// TIA Portal project "练习_V17" (V17)

(* hardware
DEVICE "S7-1200 station_1"  S7-1200 Station
   slot 0: "Rack_0"  S7-1200 Rack  Rack  V1.0
   slot 1: "PLC_1"  CPU 1215C DC/DC/DC  6ES7 215-1AG40-0XB0  V4.2
*)

// ===== PLC "PLC_1"  CPU 1215C DC/DC/DC =====

VAR_GLOBAL   // PLC tag table "默认变量表"
   "Q0.2" AT %Q0.2 : Bool;
   "Q0.3" AT %Q0.3 : Bool;
   "Q0.4" AT %Q0.4 : Bool;
   "Q0.5" AT %Q0.5 : Bool;
   "M2.4" AT %M2.4 : Bool;
   "M2.5" AT %M2.5 : Bool;
   "M2.6" AT %M2.6 : Bool;
   "M2.7" AT %M2.7 : Bool;
   "M3.0" AT %M3.0 : Bool;
   "M3.1" AT %M3.1 : Bool;
   "M3.2" AT %M3.2 : Bool;
   "M3.3" AT %M3.3 : Bool;
   "M2.0" AT %M2.0 : Bool;
   "M2.1" AT %M2.1 : Bool;
   "M2.2" AT %M2.2 : Bool;
   "M2.3" AT %M2.3 : Bool;
   "Q0.0" AT %Q0.0 : Bool;
   "Q0.1" AT %Q0.1 : Bool;
   "MD100" AT %MD100 : Time;
   "MD104" AT %MD104 : Time;
   "MD10" AT %MD10 : Real;
   "MD14" AT %MD14 : Real;
   "MD18" AT %MD18 : Real;
   "MD22" AT %MD22 : Real;
   "MD26" AT %MD26 : Real;
   "System_Byte" AT %MB1 : Byte;
   "FirstScan" AT %M1.0 : Bool;
   "DiagStatusUpdate" AT %M1.1 : Bool;
   "AlwaysTRUE" AT %M1.2 : Bool;
   "AlwaysFALSE" AT %M1.3 : Bool;
   "Clock_Byte" AT %MB0 : Byte;
   "Clock_10Hz" AT %M0.0 : Bool;
   "Clock_5Hz" AT %M0.1 : Bool;
   "Clock_2.5Hz" AT %M0.2 : Bool;
   "Clock_2Hz" AT %M0.3 : Bool;
   "Clock_1.25Hz" AT %M0.4 : Bool;
   "Clock_1Hz" AT %M0.5 : Bool;
   "Clock_0.625Hz" AT %M0.6 : Bool;
   "Clock_0.5Hz" AT %M0.7 : Bool;
   "MW30" AT %MW30 : UInt;
   "MW32" AT %MW32 : UInt;
   "MW34" AT %MW34 : UInt;
   "MW36" AT %MW36 : Int;
   "MW38" AT %MW38 : Int;
   "MW40" AT %MW40 : Int;
   "轴_3_方向" AT %Q0.6 : Bool;
   "轴_4_方向" AT %Q0.7 : Bool;
END_VAR

TYPE "运动轴"
   STRUCT
      输入 : Struct
         "IN:轴使能" : Bool := false;
         "IN:轴复位" : Bool := false;
         "IN:轴回原" : Bool := false;
         "IN:停轴" : Bool := false;
         "IN:绝对定位开" : Bool := false;
         "IN:相对定位开" : Bool := false;
         "IN:手动向前" : Bool := false;
         "IN:手动向后" : Bool := false;
         "IN:绝对目标位置" : Real := 0.0;
         "IN:相对目标位置" : Real := 0.0;
         "IN:绝对定位速度" : Real := 0.0;
         "IN:相对定位速度" : Real := 0.0;
         "IN:手动速度" : Real := 0.0;
      END_STRUCT;
      输出 : Struct
         轴使能状态 : Bool := false;
         轴错误 : Bool := false;
         轴复位完成 : Bool := false;
         轴回原完成 : Bool := false;
         轴回原中 : Bool := false;
         轴回原完成通知 : Bool := false;
         轴暂停中 : Bool := false;
         轴绝对定位完成 : Bool := false;
         轴绝对定位中 : Bool := false;
         轴相对定位完成 : Bool := false;
         轴相对定位中 : Bool := false;
         轴手动行走完成 : Bool := false;
         轴手动行走中 : Bool := false;
         轴错误代码 : Word := 16#0;
         轴错误详情 : Word := 16#0;
      END_STRUCT;
   END_STRUCT;
END_TYPE

// folder: 10-运动控制

DATA_BLOCK "轴控制_DB"   // DB13
{ S7_Optimized_Access := 'TRUE' }
VERSION : 0.1
// stored: InstanceOfName 轴控制
"轴控制"
BEGIN
END_DATA_BLOCK

DATA_BLOCK "运动轴数据"   // DB14
{ S7_Optimized_Access := 'FALSE' }
VERSION : 0.1
   VAR
      轴1 : "运动轴";
      轴2 : "运动轴";
      轴3 : "运动轴";
      轴4 : "运动轴";
   END_VAR
BEGIN
END_DATA_BLOCK

// folder: 20-报警

DATA_BLOCK "报警模块_DB"   // DB22
{ S7_Optimized_Access := 'TRUE' }
VERSION : 0.1
// stored: InstanceOfName 报警灯
"报警灯"
BEGIN
END_DATA_BLOCK

// folder: (top level)

DATA_BLOCK "轴_1"   // DB1, Motion_DB
{ S7_Optimized_Access := 'TRUE' }
AUTHOR : SIMATIC
FAMILY : BasicMC
NAME : TO_PosAx
VERSION : 6.0
// stored: InstanceOfName TO_PositioningAxis
"TO_PositioningAxis"
BEGIN
   // Axis.OnlinePtoModeCU = 16#0000_0002
   // Axis.DirectionOutputEnabledCU = TRUE
   // Axis.SelectedChannel2EnumCU = %Q0.4
   // Axis.SelectedChannel1EnumCU = %Q0.0
   // Pulse.MinDeltaDeltaFrequencyCU = 0.004
   // Pulse.MaxDeltaDeltaFrequencyCU = 1.0E+10
   // Pulse.MinDeltaFrequencyCU = 0.005
   // Pulse.MaxDeltaFrequencyCU = 9.5E+9
   // Pulse.MinFrequencyCU = 1.0
   // Pulse.MaxFrequencyCU = 100000.0
   // Pulse.OutputSourceCU = 16#0000_0000
   // Axis.SelectPTO = 0
END_DATA_BLOCK

DATA_BLOCK "轴_2"   // DB2, Motion_DB
{ S7_Optimized_Access := 'TRUE' }
AUTHOR : SIMATIC
FAMILY : BasicMC
NAME : TO_PosAx
VERSION : 6.0
// stored: InstanceOfName TO_PositioningAxis
"TO_PositioningAxis"
BEGIN
   // Axis.OnlinePtoModeCU = 16#0000_0002
   // Axis.DirectionOutputEnabledCU = TRUE
   // Axis.SelectedChannel2EnumCU = %Q0.5
   // Axis.SelectedChannel1EnumCU = %Q0.1
   // Pulse.MinDeltaDeltaFrequencyCU = 0.004
   // Pulse.MaxDeltaDeltaFrequencyCU = 1.0E+10
   // Pulse.MinDeltaFrequencyCU = 0.005
   // Pulse.MaxDeltaFrequencyCU = 9.5E+9
   // Pulse.MinFrequencyCU = 1.0
   // Pulse.MaxFrequencyCU = 100000.0
   // Pulse.OutputSourceCU = 16#0000_0000
   // Axis.SelectPTO = 1
   // Axis.OnlinePtoIndexCU = 1
END_DATA_BLOCK

DATA_BLOCK "轴_3"   // DB3, Motion_DB
{ S7_Optimized_Access := 'TRUE' }
AUTHOR : SIMATIC
FAMILY : BasicMC
NAME : TO_PosAx
VERSION : 6.0
// stored: InstanceOfName TO_PositioningAxis
"TO_PositioningAxis"
BEGIN
   // Axis.OnlinePtoModeCU = 16#0000_0002
   // Axis.DirectionOutputEnabledCU = TRUE
   // Axis.SelectedChannel2EnumCU = %Q0.6
   // Axis.SelectedChannel1EnumCU = %Q0.2
   // Pulse.MinDeltaDeltaFrequencyCU = 0.004
   // Pulse.MaxDeltaDeltaFrequencyCU = 1.0E+10
   // Pulse.MinDeltaFrequencyCU = 0.005
   // Pulse.MaxDeltaFrequencyCU = 9.5E+9
   // Pulse.MinFrequencyCU = 1.0
   // Pulse.MaxFrequencyCU = 100000.0
   // Pulse.OutputSourceCU = 16#0000_0000
   // Axis.SelectPTO = 2
   // Axis.OnlinePtoIndexCU = 2
END_DATA_BLOCK

DATA_BLOCK "轴_4"   // DB4, Motion_DB
{ S7_Optimized_Access := 'TRUE' }
AUTHOR : SIMATIC
FAMILY : BasicMC
NAME : TO_PosAx
VERSION : 6.0
// stored: InstanceOfName TO_PositioningAxis
"TO_PositioningAxis"
BEGIN
   // Axis.OnlinePtoModeCU = 16#0000_0002
   // Axis.DirectionOutputEnabledCU = TRUE
   // Axis.SelectedChannel2EnumCU = %Q0.7
   // Axis.SelectedChannel1EnumCU = %Q0.3
   // Pulse.MinDeltaDeltaFrequencyCU = 0.004
   // Pulse.MaxDeltaDeltaFrequencyCU = 1.0E+10
   // Pulse.MinDeltaFrequencyCU = 0.005
   // Pulse.MaxDeltaFrequencyCU = 9.5E+9
   // Pulse.MinFrequencyCU = 1.0
   // Pulse.MaxFrequencyCU = 100000.0
   // Pulse.OutputSourceCU = 16#0000_0000
   // Axis.SelectPTO = 3
   // Axis.OnlinePtoIndexCU = 3
END_DATA_BLOCK

ORGANIZATION_BLOCK "Main"   // OB1, LAD, ProgramCycle
TITLE = "Main Program Sweep (Cycle)"
{ S7_Optimized_Access := 'TRUE' }
VERSION : 0.1
   VAR_INPUT
      Initial_Call : Bool;   // Initial call of this OB
      Remanence : Bool;   // =True, if remanent data are available
   END_VAR
BEGIN

REGION Network 2
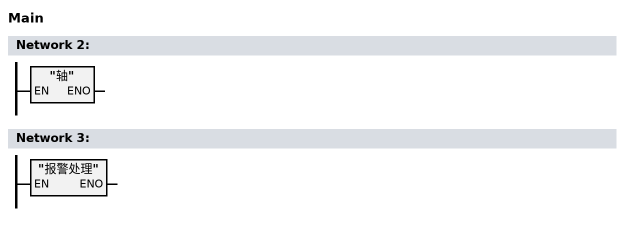
   RUNG wire#powerrail
      "轴"()
   END_RUNG
   // the same network as SCL:
   "轴"();
END_REGION

REGION Network 3
   RUNG wire#powerrail
      "报警处理"()
   END_RUNG
   // the same network as SCL:
   "报警处理"();
END_REGION
END_ORGANIZATION_BLOCK

// folder: 10-运动控制

FUNCTION_BLOCK "轴底层"   // FB11, LAD
{ S7_Optimized_Access := 'TRUE' }
VERSION : 0.1
   VAR_INPUT
      "IN:轴使能" : Bool;
      "IN:轴复位" : Bool;
      "IN:轴回原" : Bool;
      "IN:停轴" : Bool;
      "IN:绝对定位开" : Bool;
      "IN:相对定位开" : Bool;
      "IN:手动向前" : Bool;
      "IN:手动向后" : Bool;
      "IN:绝对目标位置" : Real;
      "IN:相对目标位置" : Real;
      "IN:绝对定位速度" : Real;
      "IN:相对定位速度" : Real;
      "IN:手动速度" : Real;
   END_VAR
   VAR_OUTPUT
      轴使能状态 : Bool;
      轴错误 : Bool;
      轴复位完成 : Bool;
      轴回原完成 : Bool;
      轴回原中 : Bool;
      轴回原完成通知 : Bool;
      轴暂停中 : Bool;
      轴绝对定位完成 : Bool;
      轴绝对定位中 : Bool;
      轴相对定位完成 : Bool;
      轴相对定位中 : Bool;
      轴手动行走完成 : Bool;
      轴手动行走中 : Bool;
      轴错误代码 : Word;
      轴错误详情 : Word;
   END_VAR
   VAR_IN_OUT
      轴 : TO_Axis;
      速度轴 : TO_SpeedAxis;
      定位轴 : TO_PositioningAxis;
   END_VAR
   VAR
      轴使能块 : MC_Power;
      轴复位块 : MC_Reset;
      轴回原块 : MC_Home;
      轴停止块 : MC_Halt;
      轴绝对定位块 : MC_MoveAbsolute;
      轴相对定位快 : MC_MoveRelative;
      轴手动 : MC_MoveJog;
      错误1 : Bool;
      错误2 : Bool;
      错误3 : Bool;
      错误4 : Bool;
      错误5 : Bool;
      错误6 : Bool;
      错误7 : Bool;
   END_VAR
BEGIN

REGION Network 1: 使能
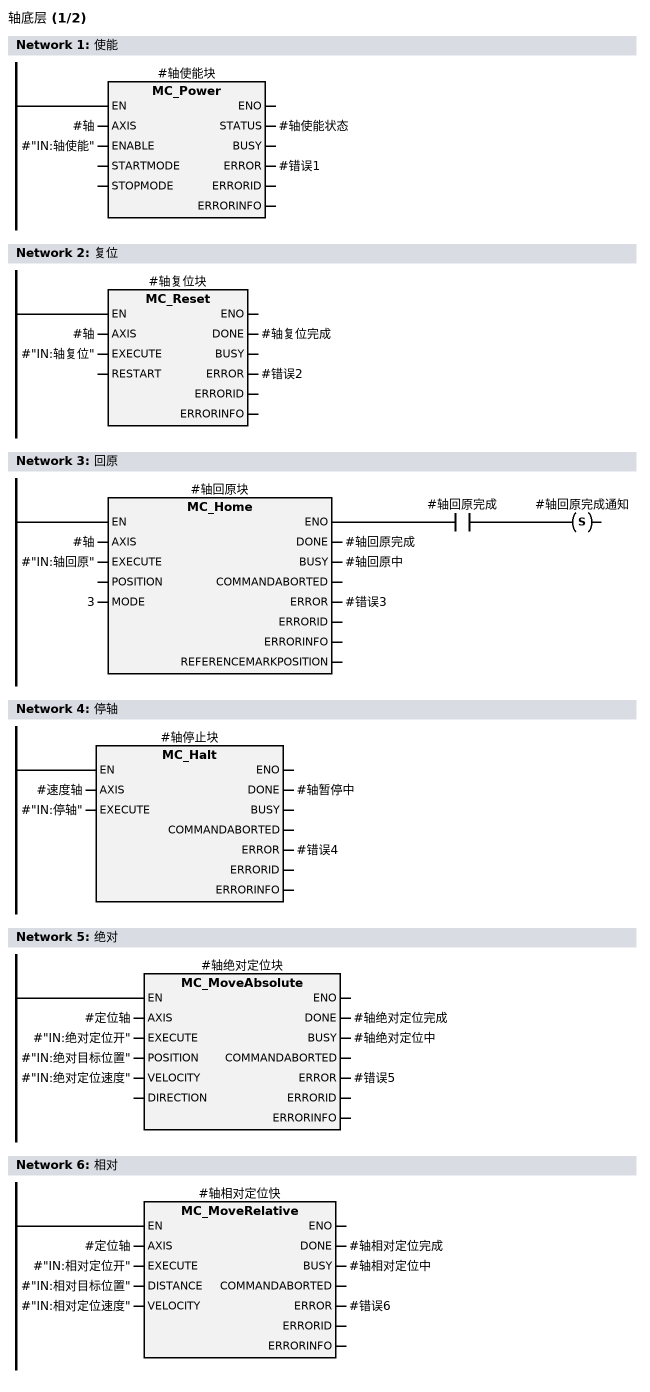
   #轴使能块(Axis := #轴, Enable := #"IN:轴使能", Status => #轴使能状态, Error => #错误1);   // MC_Power
END_REGION

REGION Network 2: 复位
   #轴复位块(Axis := #轴, Execute := #"IN:轴复位", Done => #轴复位完成, Error => #错误2);   // MC_Reset
END_REGION

REGION Network 3: 回原
   // ENO of a box is taken as its EN; it also drops when the box reports an error
   #轴回原块(Axis := #轴, Execute := #"IN:轴回原", Mode := 3, Done => #轴回原完成, Busy => #轴回原中, Error => #错误3);   // MC_Home
   IF #轴回原完成 THEN #轴回原完成通知 := TRUE; END_IF;
END_REGION

REGION Network 4: 停轴
   #轴停止块(Axis := #速度轴, Execute := #"IN:停轴", Done => #轴暂停中, Error => #错误4);   // MC_Halt
END_REGION

REGION Network 5: 绝对
   #轴绝对定位块(Axis := #定位轴,   // MC_MoveAbsolute
           Execute := #"IN:绝对定位开",
           Position := #"IN:绝对目标位置",
           Velocity := #"IN:绝对定位速度",
           Done => #轴绝对定位完成,
           Busy => #轴绝对定位中,
           Error => #错误5);
END_REGION

REGION Network 6: 相对
   #轴相对定位快(Axis := #定位轴,   // MC_MoveRelative
           Execute := #"IN:相对定位开",
           Distance := #"IN:相对目标位置",
           Velocity := #"IN:相对定位速度",
           Done => #轴相对定位完成,
           Busy => #轴相对定位中,
           Error => #错误6);
END_REGION

REGION Network 7: 手动
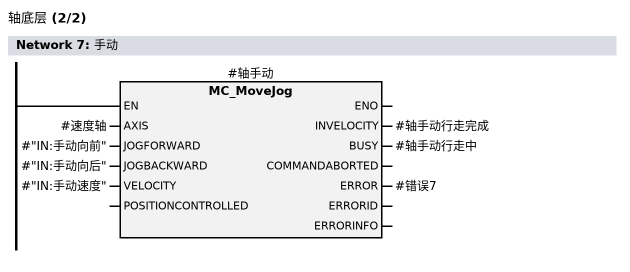
   #轴手动(Axis := #速度轴,   // MC_MoveJog
        JogForward := #"IN:手动向前",
        JogBackward := #"IN:手动向后",
        Velocity := #"IN:手动速度",
        InVelocity => #轴手动行走完成,
        Busy => #轴手动行走中,
        Error => #错误7);
END_REGION

REGION Network 8 (SCL): 轴错误
   #轴错误 := #错误1 OR #错误2 OR
              #错误3 OR #错误4 OR #错误5 OR
              #错误6 OR #错误7;
END_REGION
END_FUNCTION_BLOCK

FUNCTION_BLOCK "轴控制"   // FB12, LAD
{ S7_Optimized_Access := 'TRUE' }
VERSION : 0.1
   VAR
      轴1 : "轴底层";
      轴2 : "轴底层";
      轴3 : "轴底层";
      轴4 : "轴底层";
   END_VAR
BEGIN

REGION Network 1: 轴1控制
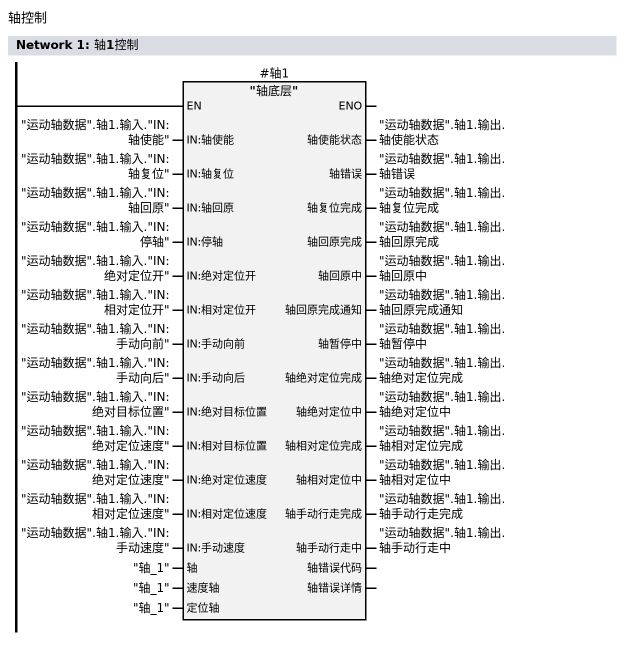
   RUNG wire#powerrail
      #轴1("IN:轴使能" := "运动轴数据".轴1.输入."IN:轴使能", "IN:轴复位" := "运动轴数据".轴1.输入."IN:轴复位", "IN:轴回原" := "运动轴数据".轴1.输入."IN:轴回原", "IN:停轴" := "运动轴数据".轴1.输入."IN:停轴", "IN:绝对定位开" := "运动轴数据".轴1.输入."IN:绝对定位开", "IN:相对定位开" := "运动轴数据".轴1.输入."IN:相对定位开", "IN:手动向前" := "运动轴数据".轴1.输入."IN:手动向前", "IN:手动向后" := "运动轴数据".轴1.输入."IN:手动向后", "IN:绝对目标位置" := "运动轴数据".轴1.输入."IN:绝对目标位置", "IN:相对目标位置" := "运动轴数据".轴1.输入."IN:绝对定位速度", "IN:绝对定位速度" := "运动轴数据".轴1.输入."IN:绝对定位速度", "IN:相对定位速度" := "运动轴数据".轴1.输入."IN:相对定位速度", "IN:手动速度" := "运动轴数据".轴1.输入."IN:手动速度", 轴 := "轴_1", 速度轴 := "轴_1", 定位轴 := "轴_1", 轴使能状态 => "运动轴数据".轴1.输出.轴使能状态, 轴错误 => "运动轴数据".轴1.输出.轴错误, 轴复位完成 => "运动轴数据".轴1.输出.轴复位完成, 轴回原完成 => "运动轴数据".轴1.输出.轴回原完成, 轴回原中 => "运动轴数据".轴1.输出.轴回原中, 轴回原完成通知 => "运动轴数据".轴1.输出.轴回原完成通知, 轴暂停中 => "运动轴数据".轴1.输出.轴暂停中, 轴绝对定位完成 => "运动轴数据".轴1.输出.轴绝对定位完成, 轴绝对定位中 => "运动轴数据".轴1.输出.轴绝对定位中, 轴相对定位完成 => "运动轴数据".轴1.输出.轴相对定位完成, 轴相对定位中 => "运动轴数据".轴1.输出.轴相对定位中, 轴手动行走完成 => "运动轴数据".轴1.输出.轴手动行走完成, 轴手动行走中 => "运动轴数据".轴1.输出.轴手动行走中, 轴错误代码 =>, 轴错误详情 =>)
   END_RUNG
   // the same network as SCL:
   #轴1("IN:轴使能" := "运动轴数据".轴1.输入."IN:轴使能",   // "轴底层"
       "IN:轴复位" := "运动轴数据".轴1.输入."IN:轴复位",
       "IN:轴回原" := "运动轴数据".轴1.输入."IN:轴回原",
       "IN:停轴" := "运动轴数据".轴1.输入."IN:停轴",
       "IN:绝对定位开" := "运动轴数据".轴1.输入."IN:绝对定位开",
       "IN:相对定位开" := "运动轴数据".轴1.输入."IN:相对定位开",
       "IN:手动向前" := "运动轴数据".轴1.输入."IN:手动向前",
       "IN:手动向后" := "运动轴数据".轴1.输入."IN:手动向后",
       "IN:绝对目标位置" := "运动轴数据".轴1.输入."IN:绝对目标位置",
       "IN:相对目标位置" := "运动轴数据".轴1.输入."IN:绝对定位速度",
       "IN:绝对定位速度" := "运动轴数据".轴1.输入."IN:绝对定位速度",
       "IN:相对定位速度" := "运动轴数据".轴1.输入."IN:相对定位速度",
       "IN:手动速度" := "运动轴数据".轴1.输入."IN:手动速度",
       轴 := "轴_1",
       速度轴 := "轴_1",
       定位轴 := "轴_1",
       轴使能状态 => "运动轴数据".轴1.输出.轴使能状态,
       轴错误 => "运动轴数据".轴1.输出.轴错误,
       轴复位完成 => "运动轴数据".轴1.输出.轴复位完成,
       轴回原完成 => "运动轴数据".轴1.输出.轴回原完成,
       轴回原中 => "运动轴数据".轴1.输出.轴回原中,
       轴回原完成通知 => "运动轴数据".轴1.输出.轴回原完成通知,
       轴暂停中 => "运动轴数据".轴1.输出.轴暂停中,
       轴绝对定位完成 => "运动轴数据".轴1.输出.轴绝对定位完成,
       轴绝对定位中 => "运动轴数据".轴1.输出.轴绝对定位中,
       轴相对定位完成 => "运动轴数据".轴1.输出.轴相对定位完成,
       轴相对定位中 => "运动轴数据".轴1.输出.轴相对定位中,
       轴手动行走完成 => "运动轴数据".轴1.输出.轴手动行走完成,
       轴手动行走中 => "运动轴数据".轴1.输出.轴手动行走中);
END_REGION

REGION Network 2 (SCL): 轴2控制
   #轴2("IN:轴使能":="运动轴数据".轴2.输入."IN:轴使能",
       "IN:轴复位":="运动轴数据".轴2.输入."IN:轴复位",
       "IN:轴回原":="运动轴数据".轴2.输入."IN:轴回原",
       "IN:停轴":="运动轴数据".轴2.输入."IN:停轴",
       "IN:绝对定位开":="运动轴数据".轴2.输入."IN:绝对定位开",
       "IN:相对定位开":="运动轴数据".轴2.输入."IN:相对定位开",
       "IN:手动向前":="运动轴数据".轴2.输入."IN:手动向前",
       "IN:手动向后":="运动轴数据".轴2.输入."IN:手动向后",
       "IN:绝对目标位置":="运动轴数据".轴2.输入."IN:绝对目标位置",
       "IN:相对目标位置":="运动轴数据".轴2.输入."IN:相对目标位置",
       "IN:绝对定位速度":="运动轴数据".轴2.输入."IN:绝对定位速度",
       "IN:相对定位速度":="运动轴数据".轴2.输入."IN:相对定位速度",
       "IN:手动速度":="运动轴数据".轴2.输入."IN:手动速度",
       轴使能状态=>"运动轴数据".轴2.输出.轴使能状态,
       轴错误=>"运动轴数据".轴2.输出.轴错误,
       轴复位完成=>"运动轴数据".轴2.输出.轴复位完成,
       轴回原完成=>"运动轴数据".轴2.输出.轴回原完成,
       轴回原中=>"运动轴数据".轴2.输出.轴回原中,
       轴回原完成通知=>"运动轴数据".轴2.输出.轴回原完成通知,
       轴暂停中=>"运动轴数据".轴2.输出.轴暂停中,
       轴绝对定位完成=>"运动轴数据".轴2.输出.轴绝对定位完成,
       轴绝对定位中=>"运动轴数据".轴2.输出.轴绝对定位中,
       轴相对定位完成=>"运动轴数据".轴2.输出.轴相对定位完成,
       轴相对定位中=>"运动轴数据".轴2.输出.轴相对定位中,
       轴手动行走完成=>"运动轴数据".轴2.输出.轴手动行走完成,
       轴手动行走中=>"运动轴数据".轴2.输出.轴手动行走中,
       轴:="轴_2",
       速度轴:="轴_2",
       定位轴:="轴_2");
END_REGION
END_FUNCTION_BLOCK

FUNCTION "轴" : Void   // FC10, LAD
{ S7_Optimized_Access := 'TRUE' }
VERSION : 0.1
BEGIN

REGION Network 1
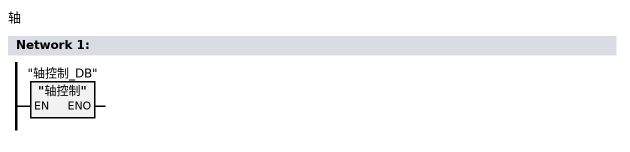
   RUNG wire#powerrail
      "轴控制_DB"()
   END_RUNG
   // the same network as SCL:
   "轴控制_DB"();   // "轴控制"
END_REGION
END_FUNCTION

// folder: 20-报警

FUNCTION_BLOCK "报警灯"   // FB21, LAD
{ S7_Optimized_Access := 'TRUE' }
VERSION : 0.1
   VAR_INPUT
      手动状态 : Bool;
      自动状态 : Bool;
      故障中 : Bool;
      自动暂停中 : Bool;
   END_VAR
   VAR_OUTPUT
      黄灯 : Bool;
      绿灯 : Bool;
      红灯 : Bool;
      蜂鸣 : Bool;
   END_VAR
BEGIN

REGION Network 1
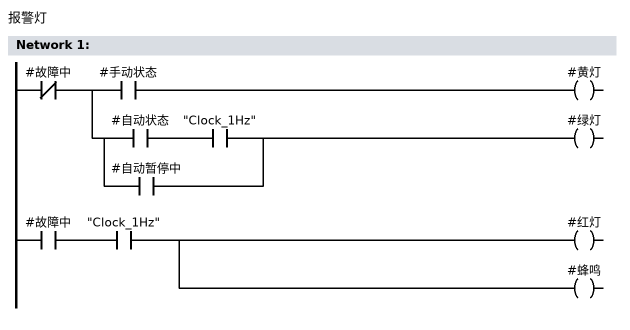
   RUNG wire#powerrail
      I_Contact( #故障中 )
      wire#w1
      Contact( #手动状态 )
      Coil( #黄灯 )
   END_RUNG
   RUNG wire#w1
      Contact( #自动状态 )
      Contact( "Clock_1Hz" )
      wire#w2
      Coil( #绿灯 )
   END_RUNG
   RUNG wire#w1
      Contact( #自动暂停中 )
   END_RUNG wire#w2
   RUNG wire#powerrail
      Contact( #故障中 )
      Contact( "Clock_1Hz" )
      wire#w3
      Coil( #红灯 )
   END_RUNG
   RUNG wire#w3
      Coil( #蜂鸣 )
   END_RUNG
   // the same network as SCL:
   #黄灯 := NOT #故障中 AND #手动状态;
   #绿灯 := NOT #故障中 AND ((#自动状态 AND "Clock_1Hz") OR #自动暂停中);
   #红灯 := #故障中 AND "Clock_1Hz";
   #蜂鸣 := #红灯;
END_REGION
END_FUNCTION_BLOCK

FUNCTION_BLOCK "报警模块"   // FB23, LAD
{ S7_Optimized_Access := 'TRUE' }
VERSION : 0.1
BEGIN
END_FUNCTION_BLOCK

FUNCTION "报警处理" : Void   // FC20, LAD
{ S7_Optimized_Access := 'TRUE' }
VERSION : 0.1
BEGIN

REGION Network 1
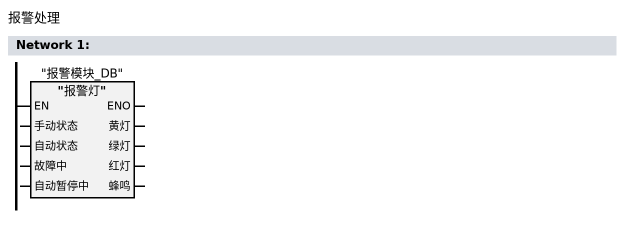
   RUNG wire#powerrail
      "报警模块_DB"(手动状态 :=, 自动状态 :=, 故障中 :=, 自动暂停中 :=, 黄灯 =>, 绿灯 =>, 红灯 =>, 蜂鸣 =>)
   END_RUNG
   // the same network as SCL:
   "报警模块_DB"();   // "报警灯"
END_REGION
END_FUNCTION